TYPE UDT_EVENT :
STRUCT
	ID: ARRAY[1..256] OF BOOL;
END_STRUCT
END_TYPE

(* stored: Version 1.1.0.1, ProductVersion 3.1.4022.16
   DUT UDT_EVENT: Id {b410adca-be06-4741-bc62-e7619bd6c0cd} *)
